{attribute 'GeneratedUsingTerminal: EL9110-0000-0016'}
{attribute addProperty BoxType "EL9110-0000-0016"}
{attribute addProperty Id "PowerOKAT %I*PowerOK_830843C11WcStateAT %I*WcState_9091E0EB2InfoDataAT %I*InfoData_6F19DB2B2"}
{attribute addProperty CRC "765678590"}
{attribute addProperty Size "5"}
TYPE EL9110_2DA353FE EXTENDS EtcSlaveTerminalBase_947E5A46 :
STRUCT
	{attribute addProperty Name "PowerOK"}
	PowerOK : PowerOK_830843C1;
	{attribute addProperty Name "WcState"}
	WcState : WcState_9091E0EB;
	{attribute addProperty Name "InfoData"}
	InfoData : InfoData_6F19DB2B;
END_STRUCT
END_TYPE

(* stored: Version 1.2.0.0, ProductVersion 3.1.4024.9
   DUT EL9110_2DA353FE: Id {1d75c39f-125f-48cf-899f-067a0ab63f20} *)
